FUNCTION_BLOCK FB_SimulatedDigOut IMPLEMENTS ITF_DigOut
VAR
	internalState : BOOL := FALSE;
END_VAR

METHOD set : BOOL
VAR_INPUT
	state : BOOL;
END_VAR
internalState := state;
END_METHOD

END_FUNCTION_BLOCK

(* stored: Version 1.1.0.1, ProductVersion 3.1.4026.8
   POU FB_SimulatedDigOut: Id {e7465166-7df2-484b-8c65-5063e075f75b}, SpecialFunc None
   Method set: Id {007f49f7-25b6-41f1-8953-09f7abb4f181} *)
